// Mitsubishi GX Works2 project: call_retEx01   PLC: Q02/Q02H

PROGRAM MAIN
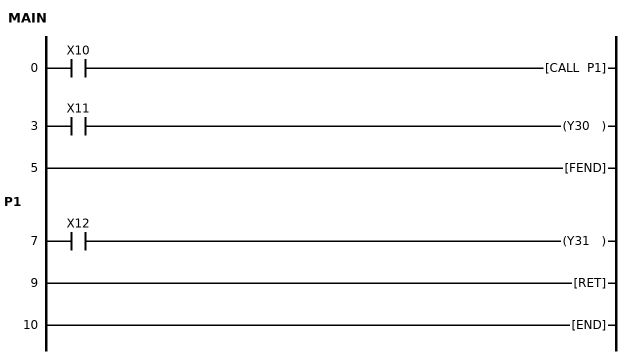
0     LD      X10
      CALL    P1
3     LD      X11
      OUT     Y30
5     FEND
      P1
7     LD      X12
      OUT     Y31
9     RET
10    END
END_PROGRAM
